{attribute 'hide_all_locals'}
(*The function block executes the drive specific homing of the axis and saves the reference in the Drive contorller*)
FUNCTION_BLOCK STOBER_MC_HOME
VAR_INPUT
	Execute					:BOOL;				(*Start homing procedure with rising edge*)
	SetModeOfOperation		:SINT:=8;
END_VAR
VAR_OUTPUT
	Done					:BOOL;				(*Homing is done Successfully*)
	ModeOfOperation	AT %Q*	:SINT;				(*output of modes of operation to be linked to the drive PDO mapping*)
	Busy					:BOOL;				(*Homing procedure is active*)
	CommandAborted			:BOOL;				(*homing procedure was aborted*)
	Error					:BOOL;				(*Error is occured*)
	ErrorID					:UDINT;				(*Error ID*)
	FBErrorID				:eERROR;			(*Function block ErrorID*)
END_VAR
VAR
	_AxisStatus					:MC_ReadStatus;
	_stStatus					:ST_AxisStatus;
	_Drivedata					:MC_ReadDriveAddress;
	stdriveadress				:ST_DriveAddress;
	_PositionLagMonitor			:ADSWRITE;
	_ExecuteTrigger				:R_TRIG;
	istate						:INT;
	_LagMonitor					:UDINT;
	init						:BOOL;
	_writeNCIOOutput			:MC_WriteNcIoOutput;
	_WriteReferenceFlag			:ADSWRITE;
	_ReferenceFlag				:UDINT;
	_AdsSetPosition				:ADSWrite;
	_stSetPosition				:st_Set_Value;
	_HomeOffSet					:DINT;
	_fbHomeOffsetCOERead		:FB_CoERead;
	_IndexID_A569				:WORD;	
	_IndexID_A516				:WORD;
	_IndexID_A586				:WORD;
	_IndexID_A542				:WORD;
	_Active						:BOOL;
	_fbHomingMethodCOERead		:FB_CoERead;
	_HomingMethod				:DINT;
	_reloop						:BOOL;
	_statusloop					:BOOL;	
	_fbCOEStatusWord_Read		:FB_CoERead;
	_StatusWord					:DINT;
	_wStatusWord				:WORD;
	_fbCOE_ModeOfOpeationDisplay:FB_CoERead;
	_ModeOfOperationDisplay		:DINT;
END_VAR
VAR_IN_OUT
	Axis						:AXIS_REF;				(*reference to axis*)
END_VAR
VAR CONSTANT
	AXISA_A569_INDEX_ID			:WORD:=16#607C;
	AXISB_A569_INDEX_ID			:WORD:=16#687C;
	AXISA_A586_INDEX_ID			:WORD:=16#6098;
	AXISB_A586_INDEX_ID			:WORD:=16#6898;
	AXISA_A516_INDEX_ID			:WORD:=16#6041;
	AXISB_A516_INDEX_ID			:WORD:=16#6841;
	AXISA_A542_INDEX_ID			:WORD:=16#6061;
	AXISB_A542_INDEX_ID			:WORD:=16#6861;
	HOMING_MODE					:SINT:=6;
END_VAR

//Write mode of operation from user input on initialisation 
IF NOT init THEN 
	ModeOfOperation:=SetModeOfOperation;
	init:=TRUE;
END_IF
IF SetModeOfOperation<>8 AND SetModeOfOperation<>9 AND SetModeOfOperation<>10 AND Execute THEN 
	Error:=TRUE;
	FBErrorID:=eERROR.WRONG_MODE;
	RETURN;		
END_IF

M_InternFbCall();
M_StateMachine();
M_GetParameterIndex();
M_OutputHandle();
M_SetPosition();

//Write mode of operation from user input if homing run is not active
IF NOT _Active THEN 
	ModeOfOperation:=SetModeOfOperation;
END_IF

//Stop the homing run if axis error comes 
IF (_AxisStatus.Error OR _AxisStatus.ErrorStop) AND _Active THEN 
	iState:=0;
	ModeOfOperation:=SetModeOfOperation;
	Error:=TRUE;
	Busy:=FALSE;
	Done:=FALSE;
	_Active:=FALSE;
END_IF

METHOD PRIVATE M_GetParameterIndex : BOOL
VAR_INPUT
END_VAR
IF stdriveadress.Channel=0 THEN 
	_IndexID_A569:=AXISA_A569_INDEX_ID;//index id for parameter A569 Axis A
	_IndexID_A586:=AXISA_A586_INDEX_ID;//index id for parameter A586 Axis A
	_IndexID_A516:=AXISA_A516_INDEX_ID;//index id for parameter A541 Axis A
	_IndexID_A542:=AXISA_A542_INDEX_ID;//index id for parameter A542 Axis A
ELSIF stdriveadress.Channel=1 THEN 
 	_IndexID_A569:=AXISB_A569_INDEX_ID;//index id for parameter A569 Axis B
	_IndexID_A586:=AXISB_A586_INDEX_ID;//Index id for parameter A586 Axis B
	_IndexID_A516:=AXISB_A516_INDEX_ID;//Index id for parameter A541 Axis B
	_IndexID_A542:=AXISB_A542_INDEX_ID;//index id for parameter A542 Axis B
END_IF
END_METHOD

METHOD PRIVATE M_InternFbCall : BOOL
VAR_INPUT
END_VAR
{warning disable C0371}	
//Read axis status 
M_ReadStatus();
//Refer to twincat NC-ADS manual index group and index offset used below in the function blocks input 
//Get Drive NC-ADS access data 
_Drivedata(	Execute:=Execute,Axis:=Axis,DriveAddress=>stdriveadress );

//Rise trigger execute trigger for function block execution 	
_ExecuteTrigger(CLK:=Execute);
	
//Enable/Disable position lag monitoring 
_PositionLagMonitor(NETID:= ,Port:=501,IDXGRP:=16#6000+stdriveadress.NcAxisId,
				IDXOFFS:=16#10,LEN:=SIZEOF(_LagMonitor),SRCADDR:=ADR(_LagMonitor),TMOUT:=T#0.1S );
				
//Overwrite NC process image--> NC control word Ctrl1			
_writeNCIOOutput(Axis:=Axis ,Device:=E_NcIoDevice.NcIoDeviceDrive , 
	NcIoOutput:=E_NcIoOutput.NcIoOutputnCtrl1,BitSelectMask:=16#10 );			

//Set reset reference flag
_WriteReferenceFlag(NETID:='',PORT:=501,IDXGRP:=16#4200+stdriveadress.NcAxisId,
					IDXOFFS:=16#1B,LEN:=SIZEOF(_ReferenceFlag),SRCADDR:=ADR(_ReferenceFlag));	

//Set target postion 
_AdsSetPosition(NETID:='',PORT:=501,IDXGRP:=16#4100+stdriveadress.NcAxisId,
				IDXOFFS:=16#60,LEN:=SIZEOF(_stSetPosition),SRCADDR:=ADR(_stSetPosition));	
				
//Read homing methods
_fbHomingMethodCOERead(	NetId:='' ,Index:=_IndexID_A586,SubIndex:=0,pDstBuf:=ADR(_HomingMethod), 
						BufLen:=SIZEOF(_HomingMethod),Axis:= Axis);	
								
//Read status word A516
_fbCOEStatusWord_Read(NetId:='',Index:=_IndexID_A516,SubIndex:=16#0,Axis:=Axis,pDstBuf:=ADR(_StatusWord),
					 BufLen:=SIZEOF(_StatusWord));
											
//Read homing offset 
_fbHomeOffsetCOERead(NetId:= ,Index:=_IndexID_A569 ,SubIndex:=0 ,pDstBuf:= ADR(_HomeOffSet),
					 BufLen:=SIZEOF(_HomeOffSet) ,Axis:= Axis);		

//Read mode of operation display 
_fbCOE_ModeOfOpeationDisplay(NetId:='',Index:=_IndexID_A542,SubIndex:=0,pDstBuf:=ADR(_ModeOfOperationDisplay),
							 BufLen:=SIZEOF(_ModeOfOperationDisplay),Axis:=Axis);
END_METHOD

METHOD PRIVATE M_OutputHandle : BOOL
VAR_INPUT
END_VAR
//Reset Error when no Execute 
IF Error AND NOT Execute THEN 
	Error:=FALSE;
	ErrorId:=0;
	FBErrorID:=eERROR.NO_ERROR;
END_IF
//Reset Done if no execute 
IF Done AND NOT Execute THEN 
	Done:=FALSE;
END_IF
//Reset Commandaborted if no execute 
IF CommandAborted AND NOT Execute THEN 
	CommandAborted:=FALSE;
END_IF
END_METHOD

METHOD PRIVATE M_ReadStatus : BOOL
VAR_INPUT
END_VAR
{warning disable C0371}	
_AxisStatus(Axis:=Axis,Enable:=TRUE,Status=>_stStatus);
//check for motion command lock when homing is runnig and MC_Stop is executed then homing run is aborted
IF _stStatus.MotionCommandsLocked AND Busy THEN 
	CommandAborted:=TRUE;
	Busy:=FALSE;
	ModeOfOperation:=SetModeOfOperation;
	iState:=0;
END_IF

//Read the staus word A516 cyclic
IF busy AND iState>30 THEN 
	REPEAT 
		_statusloop:=FALSE;
		_fbCOEStatusWord_Read(Execute:=TRUE,Axis:=Axis);
		IF NOT _fbCOEStatusWord_Read.Busy THEN 
			_fbCOEStatusWord_Read(Execute:=FALSE,Axis:=Axis);
		END_IF
		IF  _fbCOEStatusWord_Read.Error THEN 
			_fbCOEStatusWord_Read(Execute:=FALSE,Axis:=Axis);
			Error:=TRUE;
			ErrorID:=_fbCOEStatusWord_Read.AdsErrId;
			iState:=900;
			EXIT;
		END_IF		
		
	UNTIL NOT _statusloop
	END_REPEAT
ELSE 
	_fbCOEStatusWord_Read(Execute:=FALSE,Axis:=Axis);	
END_IF

//abort command if axis enable is withdrawn during homing run 
_wStatusWord:=DINT_TO_WORD(_StatusWord);
IF Busy AND _wStatusWord.1=FALSE AND iState>50 THEN 
	CommandAborted:=TRUE;
	Busy:=FALSE;
	ModeOfOperation:=SetModeOfOperation;
	iState:=0;
END_IF
END_METHOD

METHOD PRIVATE M_SetPosition : BOOL
VAR_INPUT
END_VAR

VAR
	
END_VAR
{warning disable C0371}	
//Write target position during homing mode 
IF Busy AND iState>50 THEN 
	REPEAT 
		_reloop:=FALSE;
		_stSetPosition.SetPosition:=Axis.NcToPlc.ActPos;
		
		_AdsSetPosition(WRITE:=TRUE);
		IF NOT _AdsSetPosition.busy THEN 
			_AdsSetPosition(WRITE:=FALSE);
		END_IF
		IF _AdsSetPosition.ERR THEN 
			Error:=TRUE;
			ErrorID:=_AdsSetPosition.ERRID;
			iState:=900;
			EXIT;
		END_IF
	UNTIL NOT _reloop
	END_REPEAT	
END_IF
END_METHOD

METHOD PRIVATE M_StateMachine : BOOL
VAR_INPUT
END_VAR
{warning disable C0371}	
CASE istate OF 
	0://Reset all outputs 
		_Drivedata(Axis:=Axis,Execute:=FALSE);
		IF _ExecuteTrigger.Q THEN 
			IF _AxisStatus.Standstill THEN 
				_writeNCIOOutput.Execute:=FALSE;
				_AdsSetPosition(WRITE:=FALSE);
				_PositionLagMonitor(WRITE:=FALSE);
				_WriteReferenceFlag(WRITE:=FALSE);
				_fbHomingMethodCOERead(Axis:=Axis,Execute:=FALSE);
				_fbHomeOffsetCOERead(Execute:=FALSE ,Axis:= Axis);
				_WriteReferenceFlag(WRITE:=FALSE);	
				_fbCOEStatusWord_Read(Axis:=Axis,Execute:=FALSE);		
				Busy:=TRUE;
				_Active:=TRUE;
				Done:=FALSE;
				Error:=FALSE;
				ErrorID:=0;
				FBErrorID:=(eERROR.NO_ERROR);
				CommandAborted:=FALSE;
				iState:=iState+5;	
			ELSE
				Error:=TRUE;
				FBErrorID:=(eERROR.AXIS_NOT_ENABLED);
				istate:=900;	
			END_IF
		END_IF
	5://reset NC reference FLAG 
		_ReferenceFlag:=0;
		_WriteReferenceFlag(WRITE:=TRUE);
		IF NOT _WriteReferenceFlag.BUSY THEN 
			_WriteReferenceFlag(WRITE:=FALSE);
			iState:=iState+5;
		ELSIF _WriteReferenceFlag.ERR THEN
			Error:=TRUE;
			ErrorID:=_WriteReferenceFlag.ERRID;
			iState:=900;	
		END_IF
	
	10://Get the drive NC-ADS data 
		_Drivedata.Execute:=TRUE;
		IF NOT _Drivedata.Busy AND _Drivedata.Done THEN
			iState:=iState+10;
		END_IF 	
		IF _Drivedata.Error THEN 
			Error:=TRUE;
			iState:=900;
		END_IF
		
	20://Disable Position lag monitoring
		_LagMonitor:=0;
		_PositionLagMonitor(WRITE:=TRUE);
		IF NOT 	_PositionLagMonitor.BUSY THEN
			_PositionLagMonitor(WRITE:=FALSE);
			iState:=iState+10;
		ELSIF 	_PositionLagMonitor.ERR THEN 
			Error:=TRUE;
			ErrorID:=_PositionLagMonitor.ERRID;
			iState:=900;
		END_IF
		
	30: //set Mode of operation to homing mode 
			ModeOfOperation:=HOMING_MODE;	
			istate:=istate+10;
		
	40://confirm mode of operation 	
		_fbCOE_ModeOfOpeationDisplay(Execute:=TRUE,Axis:=Axis);
		IF NOT _fbCOE_ModeOfOpeationDisplay.Busy THEN 
			_fbCOE_ModeOfOpeationDisplay(Execute:=FALSE,Axis:=Axis);
			IF _ModeOfOperationDisplay<>HOMING_MODE THEN 
				Error:=TRUE;
				FBErrorID:=eERROR.NO_DEVICE_LINK;
				iState:=900;
			ELSE
				iState:=iState+10;	
			END_IF
		ELSIF 	_fbCOE_ModeOfOpeationDisplay.Error THEN 
			Error:=TRUE;
			ErrorID:=_fbCOE_ModeOfOpeationDisplay.AdsErrId;
			_fbCOE_ModeOfOpeationDisplay(Execute:=FALSE,Axis:=Axis);
			iState:=900;
		END_IF
		
			
	50://Read Homing offset 
		_fbHomeOffsetCOERead(Axis:=Axis,Execute:=TRUE);
		IF NOT _fbHomeOffsetCOERead.Busy THEN 
			_fbHomeOffsetCOERead(Execute:=FALSE ,Axis:= Axis);
			istate:=istate+10;
		ELSIF _fbHomeOffsetCOERead.Error THEN 
			Error:=TRUE;
			ErrorID:=_fbHomeOffsetCOERead.AdsErrId;
			iState:=900;
		END_IF
		
	60://Read homing method 
		_fbHomingMethodCOERead(Axis:=Axis,Execute:=TRUE);			
		IF NOT _fbHomingMethodCOERead.Busy THEN 
			_fbHomingMethodCOERead(Axis:=Axis,Execute:=FALSE);
			IF (_HomingMethod=0) THEN 
				Error:=TRUE;
				FBErrorID:=(eERROR.HOMING_METHOD_INACTIVE);
				iState:=900;
			ELSE	
				iState:=iState+10;	
			END_IF
		ELSIF 	_fbHomingMethodCOERead.Error THEN
			Error:=TRUE;
			ErrorID:=_fbHomingMethodCOERead.AdsErrId;
			iState:=900;
		END_IF
	70://Reset bit 4 of NC control word and start homing
		_writeNCIOOutput.BitValues:=0;
		_writeNCIOOutput.Execute:=TRUE;
		IF _writeNCIOOutput.Done THEN
				istate:=istate+10;
				_writeNCIOOutput.Execute:=FALSE;
		END_IF		
			
	80://wait till homing is done 	or wait till bit 10 of status word is true 	
		 IF _wStatusWord.10 = TRUE AND _wStatusWord.12 THEN 
			 ModeOfOperation:=8;
			 iState:=iState+10;
		 END_IF
		
	90://Set NC reference FLAG
		 _ReferenceFlag:=1;
		_WriteReferenceFlag(WRITE:=TRUE);
		IF NOT _WriteReferenceFlag.BUSY THEN 
			_WriteReferenceFlag(WRITE:=FALSE);
			iState:=iState+10;
		ELSIF _WriteReferenceFlag.ERR THEN
			Error:=TRUE;
			ErrorID:=_WriteReferenceFlag.ERRID;
			iState:=900;	
		END_IF
	100://Enable position monitoring 
		_LagMonitor:=1;
		_PositionLagMonitor(WRITE:=TRUE);
		IF NOT 	_PositionLagMonitor.BUSY THEN
			_PositionLagMonitor(WRITE:=FALSE);
			iState:=iState+10;
		ELSIF 	_PositionLagMonitor.ERR THEN 
			Error:=TRUE;
			ErrorID:=_PositionLagMonitor.ERRID;
		END_IF	
	
	110://set mode of operation back to setoperationmode 
		ModeOfOperation:=SetModeOfOperation;
		_writeNCIOOutput.BitValues:=0;
		_writeNCIOOutput.Execute:=TRUE;
		IF _writeNCIOOutput.Done THEN 
				_writeNCIOOutput.Execute:=FALSE;
				Done:=TRUE;
				Busy:=FALSE;
				_Active:=FALSE;
				iState:=0;
		END_IF
	
	900://Error state
		istate:=0;
		ModeOfOperation:=SetModeOfOperation;
		Busy:=FALSE;
		_Active:=FALSE;
END_CASE
END_METHOD

END_FUNCTION_BLOCK

(* stored: Version 1.1.0.1, ProductVersion 3.1.4024.6
   POU STOBER_MC_HOME: Id {7089af26-30a8-48e9-be61-24acabe99986}, SpecialFunc None
   Method M_GetParameterIndex: Id {54e32b23-da6c-42fb-b7a3-0c51c43ee6e9}
   Method M_InternFbCall: Id {dfdc63eb-4c88-425c-8eee-3fd808d3fc15}
   Method M_OutputHandle: Id {669b98cf-8b34-4a83-9201-1cedc378bb93}
   Method M_ReadStatus: Id {88b8c826-f773-4afb-8119-e789e853abdc}
   Method M_SetPosition: Id {e5c91de0-c6dc-46f3-bb4b-c69e4d2f6ee9}
   Method M_StateMachine: Id {4017c47f-b8b7-4e53-8e3c-d5a9b5891d22} *)
